// Block: MES_Com_Channel_Topic4XX

DATA_BLOCK MES_Com_Channel_Topic4XX
VERSION : 0.1
   NON_RETAIN
   VAR
      RECEIVE : Struct
         ack : DInt;
         msg : MES_Msg;
      END_STRUCT;
      SEND : Struct
         ack : DInt;
         msg : MES_Msg;
      END_STRUCT;
   END_VAR

BEGIN
   // No initialization required
END_DATA_BLOCK
